// TIA Portal V17 export
// export: Created 2025-01-08T13:55:37.0815271Z, ExportSetting WithDefaults, DisplayName Totally Integrated Automation Portal, DisplayVersion V17, DisplayName TIA Portal Openness, DisplayVersion V17, DisplayName TIA Portal Version Control Interface, DisplayVersion V17, DisplayName SINAMICS Startdrive Advanced, DisplayVersion V17 Update2, DisplayName SINAMICS Startdrive G130, G150, S120, S150, SINAMICS MV, S210, DisplayVersion V17 Update2, DisplayName SINAMICS Startdrive G110M, G120, G120C, G120D, G120P, G115D, DisplayVersion V17 Update2, DisplayName STEP 7 Professional, DisplayVersion V17, DisplayName STEP 7 Safety, DisplayVersion V17, DisplayName WinCC Advanced, DisplayVersion V17
TYPE "HSMMachineParaMask4"
// stored: IsFailsafeCompliant false
   STRUCT
      "iSPS-DB-No-Stat" : Bool;
      iSignalFormat : Bool;
      iLowLabDiam : Bool;
      iCoreDiameter : Bool;
      iWebBreakRest : Bool;
      iLeverSetup : Bool;
      iLeverMinPos : Bool;
      iLeverMaxPos : Bool;
      "iUW-BufLength" : Bool;
      iTwinLabelMd : Bool;
      iLabQueuwTolerance : Bool;
      iResetEvents : Bool;
      iMaintananceDistancekm : Bool;
      iMaintananceDays : Bool;
      iProductSensorMode : Bool;
      iRewinderDiameterWarning : Bool;
   END_STRUCT;
END_TYPE
